# B&R Automation Studio project DriveControl
Automation Studio 4.5.2.102; Default project; technology packages: Acp10Arnc0 5.11.1

## Configuration SampleText

### Task classes (Cpu.sw)
```
Cyclic#4:
  Program <- Program.prg
Libraries: Acp10sdc, sys_lib, Runtime, asstring, DriveLib, Acp10man, Acp10par, NcGlobal, AsBrStr
```

### Hardware
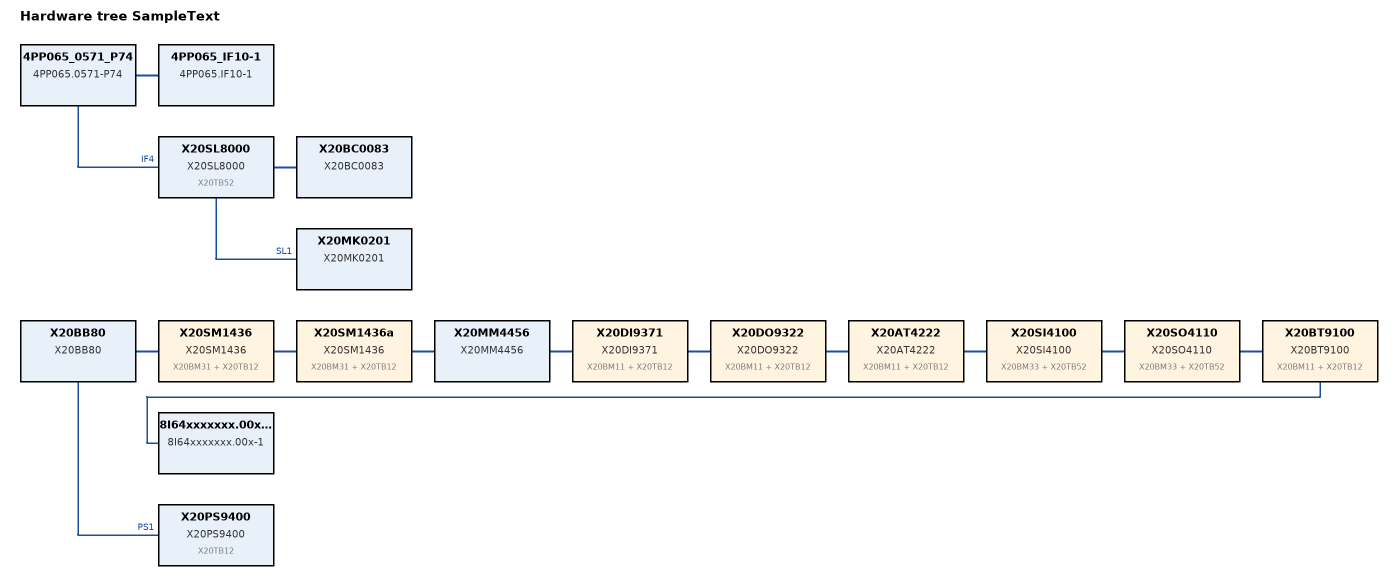
```
4PP065_0571_P74 : 4PP065.0571-P74 v1.1.2.0
  Connector IF4:
    EplInterfaceRedundant = 0
    EplEthInterfaceRedundant = 0
  Connector IF5:
    ActivateDevice = 1
    Mode = Manual
    InternetAddress = 10.1.1.13
    SubnetMask = 255.255.255.0
  ConfigurationID = labBR
  Simulation = 1
  TimerDeviceType = EPLX2X
  TimerDevice = 4PP065_0571_P74.IF4
  TaskClassIdleTime = 2000
  Cyclic1Duration = 2000
  Cyclic1Tolerance = 0
  Cyclic1Output = 1
4PP065_IF10-1 : 4PP065.IF10-1 v1.0.3.0  [SS -> 4PP065_0571_P74.SS1]
8I64xxxxxxx.00x-1 : 8I64xxxxxxx.00x-1 v1.3.9.1  [X2X1 -> X20BT9100.X2X1 [Cable Type=X2XCable, Length=10, Version=1.0.0.2]]
  FunctionModel = Standard
  packedETAD = packed
  packedETI = packed
  packedCMDD = packed
  packedCMI = packed
  UNS = 220
  NCR = 10
  NSP = 890
  COS = 64
  RSC = 33000
X20AT4222 : X20AT4222 v1.2.3.0  [SS1 -> X20TB12e.SS; SL -> X20BM11c.SL1]
X20BB80 : X20BB80 v1.0.2.0
X20BC0083 : X20BC0083 v2.8.0.0  [PLK1 -> X20SL8000.PLK2 (NodeNumber=2) [Cable Type=PowerlinkCable, Length=10, Version=1.0.0.2]; SL -> X20BB80.SL1]
X20BM11 : X20BM11 v1.0.0.1  [X2X1 -> X20BM33a.X2X2]
X20BM11a : X20BM11 v1.0.0.1  [X2X1 -> X20MM4456.X2X2]
X20BM11b : X20BM11 v1.0.0.1  [X2X1 -> X20BM11a.X2X2]
X20BM11c : X20BM11 v1.0.0.1  [X2X1 -> X20BM11b.X2X2]
X20BM31 : X20BM31 v1.0.0.1  [X2X1 -> X20BB80.IF1]
X20BM31a : X20BM31 v1.0.0.1  [X2X1 -> X20BM31.X2X2]
X20BM33 : X20BM33 v1.0.0.4  [X2X1 -> X20BM11c.X2X2]
X20BM33a : X20BM33 v1.0.0.4  [X2X1 -> X20BM33.X2X2]
X20BT9100 : X20BT9100 v1.0.3.0  [SS1 -> X20TB12f.SS; SL -> X20BM11.SL1]
X20DI9371 : X20DI9371 v1.0.2.0  [SS1 -> X20TB12c.SS; SL -> X20BM11a.SL1]
X20DO9322 : X20DO9322 v1.0.3.0  [SS1 -> X20TB12d.SS; SL -> X20BM11b.SL1]
X20MK0201 : X20MK0201 v1.0.0.0  [SL -> X20SL8000.SL1]
X20MM4456 : X20MM4456 v1.1.5.0  [X2X1 -> X20BM31a.X2X2]
X20PS9400 : X20PS9400 v1.0.2.4  [SS1 -> X20TB12.SS; PS -> X20BB80.PS1]
X20SI4100 : X20SI4100 v1.10.1.1  [SS1 -> X20TB52.SS; SL -> X20BM33.SL1]
X20SL8000 : X20SL8000 v1.6.5.1  [PLK1 -> 4PP065_0571_P74.IF4 (NodeNumber=1) [Cable Type=PowerlinkCable, Length=10, Version=1.0.0.2]; PLK2 -> X20BC0083.PLK1 (NodeNumber=1) [Cable Type=PowerlinkCable, Length=10, Version=1.0.0.2]; SS1 -> X20TB52b.SS]
  SafeProject = SafeLOGIC-1
X20SM1436 : X20SM1436 v1.4.2.1  [SS1 -> X20TB12a.SS; SL -> X20BM31.SL1]
X20SM1436a : X20SM1436 v1.4.2.1  [SS1 -> X20TB12b.SS; SL -> X20BM31a.SL1]
X20SO4110 : X20SO4110 v1.10.1.1  [SS1 -> X20TB52a.SS; SL -> X20BM33a.SL1]
  SafeModuleID = 3
X20TB12 : X20TB12 v1.0.0.0
X20TB12a : X20TB12 v1.0.0.0
X20TB12b : X20TB12 v1.0.0.0
X20TB12c : X20TB12 v1.0.0.0
X20TB12d : X20TB12 v1.0.0.0
X20TB12e : X20TB12 v1.0.0.0
X20TB12f : X20TB12 v1.0.0.0
X20TB52 : X20TB52 v1.0.0.1
X20TB52a : X20TB52 v1.0.0.1
X20TB52b : X20TB52 v1.0.0.1
```

### IoMap.iom - 4PP065_0571_P74/IoMap.iom
```iecst
VAR_CONFIG
	::Program:Drive.state AT %IW."8I64xxxxxxx.00x-1".ETAD_Input;
	::Program:Drive.command AT %QW."8I64xxxxxxx.00x-1".CMDD_Output;
	::Program:Drive.speed AT %QW."8I64xxxxxxx.00x-1".LFRD_Output;
	::Program:Door.direction AT %IX."X20DI9371".DigitalInput01;
	::Program:Door.sw1 AT %IX."X20DI9371".DigitalInput02;
	::Program:Door.sw2 AT %IX."X20DI9371".DigitalInput03;
	::Program:Door.sw3 AT %IX."X20DI9371".DigitalInput04;
	::Program:Door.sw4 AT %IX."X20DI9371".DigitalInput05;
	::Program:Led.led1 AT %QX."X20DO9322".DigitalOutput02;
	::Program:Led.led2 AT %QX."X20DO9322".DigitalOutput03;
	::Program:Led.led3 AT %QX."X20DO9322".DigitalOutput04;
	::Program:Led.led4 AT %QX."X20DO9322".DigitalOutput05;
END_VAR
```

### Acp10cfg.ncc - 4PP065_0571_P74/Motion/Acp10cfg.ncc
```
NcConfiguration (Version=5.11.1, NcSwId=Acp10)
  ACP10CF1_typ:
    cnt_nettrc_rec_drive = 150
    bufsize_trace_upload = 1200
    tc_nc_man_task = Cyclic #1
    glob_pv_as_ncobject = Yes
    ncsys_dl_broadcast = Yes
    ncsys_dl_acp_reset = Yes
    safemc_log_err_to_ax = Yes
    network_init:
      ncsw_init_execute = Yes
      automatic_execute = No
      node_nr_warning = Yes
      net_err_before_ncact = Yes
    nettrc:
      enter_parsecrec = Yes
      enter_ncaction = Yes
      save_ring_startidx = No
    cam_prof_download:
      cam_dat_dl_parallel = No
      tc_cam_dl_parallel = Task class for NC Manager task
    sdc_if[0]:
      if_name = SDC_IF1
      mc_broadcast_size = 800
      mc_broadcast_extdat = No
```

## Configuration Simulation

### Task classes (Cpu.sw)
```
Libraries: AsIecCon, astime, Acp10sdc, Acp10man, Acp10par, NcGlobal
```

## Logical view

Binary libraries used (declarations not repeated): Runtime, Operator, AsIecCon, astime, sys_lib, asstring, Acp10sdc 5.11.1, Acp10man 5.11.1, Acp10par 5.11.1, NcGlobal 5.11.1, AsBrStr

### Library Logical/Libraries/DriveLib (ANSIC)

#### Types.typ - Exported data types
```iecst
TYPE
	DriveCommands :
		(
		CMD_SWITCH_ON,
		CMD_SHUTDOWN,
		CMD_ENABLE,
		STATE_SWITCHED_ON,
		STATE_READY,
		STATE_DISABLED
		);
	DoorStates :
		(
		ST_INIT,
		ST_UNKNOWN,
		ST_OPEN,
		ST_CLOSE,
		ST_ACC_POS,
		ST_ACC_NEG,
		ST_POS,
		ST_NEG,
		ST_DEC_POS,
		ST_DEC_NEG
		);
END_TYPE
```

#### DriveLib.fun - Exported functions and function blocks
```iecst
{REDUND_ERROR} {REDUND_UNREPLICABLE} FUNCTION_BLOCK DriveStateMachine (* *) (*$GROUP=User,$CAT=User,$GROUPICON=User.png,$CATICON=User.png*)
	VAR_INPUT
		state : {REDUND_UNREPLICABLE} UINT;
		enable : {REDUND_UNREPLICABLE} BOOL;
	END_VAR
	VAR_OUTPUT
		command : {REDUND_UNREPLICABLE} UINT;
		speed : {REDUND_UNREPLICABLE} INT;
	END_VAR
END_FUNCTION_BLOCK

{REDUND_ERROR} {REDUND_UNREPLICABLE} FUNCTION_BLOCK LedStateMashine (*TODO: Add your comment here*) (*$GROUP=User,$CAT=User,$GROUPICON=User.png,$CATICON=User.png*)
	VAR_INPUT
		state : {REDUND_UNREPLICABLE} UINT;
	END_VAR
	VAR_OUTPUT
		led1 : {REDUND_UNREPLICABLE} BOOL;
		led2 : {REDUND_UNREPLICABLE} BOOL;
		led3 : {REDUND_UNREPLICABLE} BOOL;
		led4 : {REDUND_UNREPLICABLE} BOOL;
		timer : {REDUND_UNREPLICABLE} INT;
	END_VAR
END_FUNCTION_BLOCK

{REDUND_ERROR} {REDUND_UNREPLICABLE} FUNCTION_BLOCK DoorStateMashine (*TODO: Add your comment here*) (*$GROUP=User,$CAT=User,$GROUPICON=User.png,$CATICON=User.png*)
	VAR_INPUT
		state : {REDUND_UNREPLICABLE} UINT;
		sw1 : {REDUND_UNREPLICABLE} BOOL;
		sw2 : {REDUND_UNREPLICABLE} BOOL;
		sw3 : {REDUND_UNREPLICABLE} BOOL;
		sw4 : {REDUND_UNREPLICABLE} BOOL;
		direction : {REDUND_UNREPLICABLE} BOOL;
	END_VAR
	VAR_OUTPUT
		speed : {REDUND_UNREPLICABLE} INT;
	END_VAR
END_FUNCTION_BLOCK
```

#### DriveStateMachine.c
```c
#include <bur/plctypes.h>
#ifdef __cplusplus
	extern "C"
	{
#endif
	#include "DriveLib.h"
#ifdef __cplusplus
	};
#endif
void DriveStateMachine(struct DriveStateMachine* inst)
{
	/*TODO: Add your code here*/
	UINT state = inst->state & 0x6f;
	switch(state)
	{
		case STATE_DISABLED:
			if(inst->enable == 0)
				inst->command = CMD_SHUTDOWN;
			else
				inst->command = CMD_SWITCH_ON;
			break;

		case STATE_SWITCHED_ON:
			if(inst->enable == 0)
				inst->command = CMD_SHUTDOWN;
			else
				inst->command = CMD_ENABLE;
			break;

		case STATE_READY:
			if(inst->enable == 0)
				inst->command = CMD_SHUTDOWN;
			break;
	}
}
```

#### LedStateMashine.c
```c
#include <bur/plctypes.h>
#ifdef __cplusplus
	extern "C"
	{
#endif
	#include "DriveLib.h"
#ifdef __cplusplus
	};
#endif
/* TODO: Add your comment here */
void LedStateMashine(struct LedStateMashine* inst)
{
	/*TODO: Add your code here*/
	inst->timer++;
	switch(inst->state)
	{
		case ST_INIT:
			break;

		case ST_UNKNOWN:
			if(inst->timer % 10 == 0)
			{
				inst->led1 = !inst->led1;
				inst->led2 = !inst->led2;
				inst->led3 = !inst->led3;
				inst->led4 = !inst->led4;
			}
			break;

		case ST_OPEN:
			inst->led1 = 0;
			inst->led2 = 0;
			inst->led3 = 0;
			inst->led4 = 0;
			break;

		case ST_CLOSE:
			inst->led1 = 1;
			inst->led2 = 1;
			inst->led3 = 1;
			inst->led4 = 1;
			break;

		case ST_ACC_POS:
			inst->led1 = 1;
			inst->led2 = 0;
			inst->led3 = 0;
			inst->led4 = 0;
			break;

		case ST_ACC_NEG:
			inst->led1 = 1;
			inst->led2 = 1;
			inst->led3 = 1;
			inst->led4 = 0;
			break;

		case ST_POS:
			inst->led1 = 1;
			inst->led2 = 1;
			inst->led3 = 0;
			inst->led4 = 0;
			break;

		case ST_NEG:
			inst->led1 = 1;
			inst->led2 = 1;
			inst->led3 = 0;
			inst->led4 = 0;
			break;

		case ST_DEC_POS:
			inst->led1 = 1;
			inst->led2 = 1;
			inst->led3 = 1;
			inst->led4 = 0;

		case ST_DEC_NEG:
			inst->led1 = 1;
			inst->led2 = 0;
			inst->led3 = 0;
			inst->led4 = 0;
			break;
	}
}
```

#### DoorStateMashine.c
```c
#include <bur/plctypes.h>
#ifdef __cplusplus
	extern "C"
	{
#endif
	#include "DriveLib.h"
#ifdef __cplusplus
	};
#endif
/* TODO: Add your comment here */
void DoorStateMashine(struct DoorStateMashine* inst)
{
	/*TODO: Add your code here*/
	switch(inst->state)
	{
		case ST_INIT:
			inst->state = ST_UNKNOWN;
			break;

		case ST_UNKNOWN:
			if(inst->sw1 && inst->direction == 0)
				inst->state = ST_OPEN;
			if(inst->sw4 && inst->direction == 1)
				inst->state = ST_CLOSE;
		break;

		case ST_OPEN:
			inst->speed = 0;
			if(inst->direction == 0)
				inst->state = ST_ACC_POS;
			break;

		case ST_CLOSE:
			inst->speed = 0;
			if(inst->direction == 1)
				inst->state = ST_ACC_NEG;
			break;

		case ST_ACC_POS:
			inst->speed = 200;
			if(inst->sw2)
				inst->state = ST_POS;
			else if(inst->direction == 1)
				inst->state = ST_DEC_NEG;
			break;

		case ST_ACC_NEG:
			inst->speed = 0 - 200;
			if(inst->sw3)
				inst->state = ST_NEG;
			else if(inst->direction == 0)
				inst->state = ST_DEC_POS;
			break;

		case ST_POS:
			inst->speed = 600;
			if(inst->sw3)
				inst->state = ST_DEC_POS;
			else if(inst->direction == 1)
				inst->state = ST_NEG;
			break;

		case ST_NEG:
			inst->speed = -600;
			if(inst->sw2)
				inst->state = ST_DEC_NEG;
			else if(inst->direction == 0)
				inst->state = ST_POS;
			break;

		case ST_DEC_POS:
			inst->speed = 200;
			if(inst->sw4)
				inst->state = ST_CLOSE;
			break;

		case ST_DEC_NEG:
			inst->speed = 0 - 200;
			if(inst->sw1)
				inst->state = ST_OPEN;
			break;
	}
}
```

### Program Logical/Program

#### Variables.var
```iecst
VAR
	Drive : DriveStateMachine := (0);
	Door : DoorStateMashine := (0);
	Led : LedStateMashine := (0);
END_VAR
```

#### Main.c
```c
#include <bur/plctypes.h>

#ifdef _DEFAULT_INCLUDES
	#include <AsDefault.h>
#endif

void _INIT ProgramInit(void)
{
	Drive.enable = 1;
}

void _CYCLIC ProgramCyclic(void)
{
	DoorStateMashine(&Door);
	Drive.speed = Door.speed;
	DriveStateMachine(&Drive);
	Led.state = Door.state;
	LedStateMashine(&Led);
}

void _EXIT ProgramExit(void)
{

}
```

Listed in the project but not available here: Logical/Libraries/DriveLib/Constants.var
